{attribute 'reflection'}
FUNCTION_BLOCK PUBLIC FB_EncoderBase EXTENDS FB_DevBase
VAR_INPUT
END_VAR
VAR_OUTPUT
	nOutPosition		: LREAL	:= 0	; // Scaled position output
	nOutRaw				: UDINT := 0	; // Raw output value	 
	nVelocity			: LREAL	:= 0 	; // Velocity [units/sec]
END_VAR
VAR
	fPulsesPerUnit		: LREAL := 1	; // Scale factor for output [units/pulse]
	fOffset				: LREAL := 0	; // Offset for output
	bIcfInverted		: BOOL	:= FALSE; // Invert output position = standard false  
END_VAR

METHOD PUBLIC FastTask : BOOL
VAR_INPUT
END_VAR
END_METHOD

METHOD PUBLIC Init : BOOL
VAR_INPUT
	// Message location data
	nId			: UDINT ; // Identification number of object
	nParentId	: UDINT ; // Id of higher level If aplicable (0 = no parent)
	// Configuration
	fPulsesPerUnit	: LREAL	; // Scale factor for output [units/pulse]
	fOffset			: LREAL	; // Offset for output
	bIcfInverted	: BOOL	; // Invert output position = standard false  
END_VAR


// ====== Calculate device id =====
	ExecIdentifyDevice(nId,nParentId, E_ComponentTypes.Encoder);

// ====== Set manual device type ======
	eDevType := E_Devices.Encoder ;	

	
// ===== Coppy values to function memory ======
	THIS^.fPulsesPerUnit	:= MAX(fPulsesPerUnit,0.01); // Minimum value of 1
	THIS^.fOffset			:= fOffset;
	THIS^.bIcfInverted		:= bIcfInverted;
	
	
bInitOk := TRUE ;
END_METHOD

END_FUNCTION_BLOCK

(* stored: Version 1.1.0.1, ProductVersion 3.1.4024.5
   POU FB_EncoderBase: Id {78ccea55-8da3-46e5-834a-35136183596e}, SpecialFunc None
   Method FastTask: Id {0ad38990-cab6-4c8e-9e02-268fa5106cf5}
   Method Init: Id {4b96b077-08c2-0f5d-0b64-41873bbad573} *)
